KUKA KRL program: Test1.src, Test1.dat

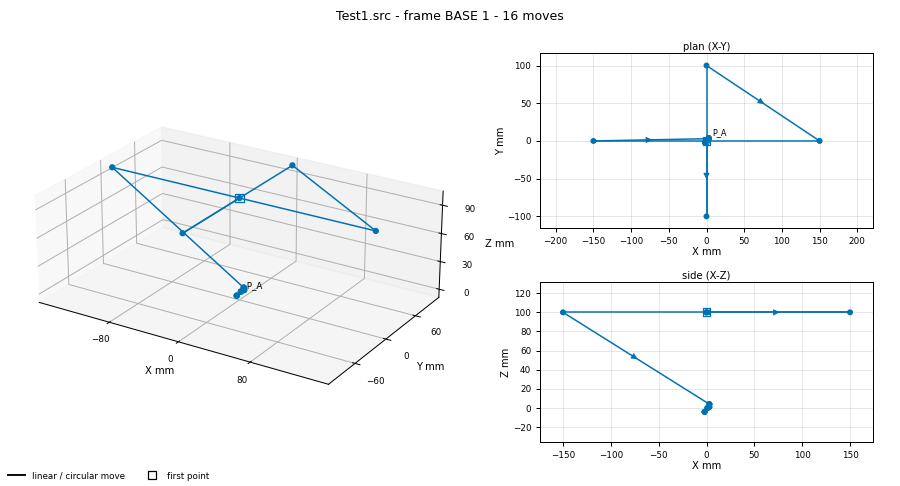
[picture p0: tool path of Test1.src in frame BASE 1, 16 of 18 moves have a stored position in this frame; points joined in program order, loops and branches not executed]
--- Test1.src ---
&ACCESS RVO1
&COMMENT Modul (src/dat) with INI line and PTP HOME at start and end of Program
DEF Test1 ( )
;FOLD INI
  ;FOLD BASISTECH INI
    GLOBAL INTERRUPT DECL 3 WHEN $STOPMESS==TRUE DO IR_STOPM ( )
    INTERRUPT ON 3
    BAS (#INITMOV,0 )
  ;ENDFOLD (BASISTECH INI)
  ;FOLD USER INI
    ;Make your modifications here

  ;ENDFOLD (USER INI)
;ENDFOLD (INI)
$TOOL = TOOL_DATA[1]
$BASE = BASE_DATA[1]

;FOLD PTP HOME  Vel= 100 % DEFAULT;%{PE}%MKUKATPBASIS,%CMOVE,%VPTP,%P 1:PTP, 2:HOME, 3:, 5:100, 7:DEFAULT
$BWDSTART = FALSE
PDAT_ACT=PDEFAULT
FDAT_ACT=FHOME
BAS (#PTP_PARAMS,100 )
$H_POS=XHOME
PTP  XHOME
;ENDFOLD

  LIN {X 0, Y 0, Z 100}
  LIN {X 0, Y -100, Z 100}
  LIN {X 0, Y 100, Z 100}
  LIN {X 150, Y 0, Z 100}
  LIN {X -150, Y 0, Z 100}

 IF mode == 1 THEN   ;IF NOT mode == 1 THEN can do it this way as well
   LIN P_A
 ELSEIF mode == 2  THEN
   LIN P_C
 ELSE
   LIN P_B
 ENDIF

   mode=2 ;change the mode during the program
 IF mode == 2 THEN
   LIN P_C
 ELSE
   LIN P_B
 ENDIF

  mode=1

 WHILE mode<4
   LIN P_A
   mode=mode + 1
 ENDWHILE

 FOR i=1 TO 3
 LIN P_D
 ENDFOR

LIN P_A
LIN P_B
LIN P_C
LIN P_D
PTP XHOME
END

--- Test1.dat ---
&ACCESS RVO1
&COMMENT Modul (src/dat) with INI line and PTP HOME at start and end of Program
DEFDAT Test1 PUBLIC

DECL INT mode = 1
DECL BOOL ready = FALSE

DECL E6POS P_A = {X 3, Y 3, Z 4, A 0, B 0, C 0}
DECL E6POS P_B = {X -2, Y -2, Z -4, A 0, B 0, C 0}
DECL E6POS P_C = {X 1, Y 1, Z 0, A 0, B 0, C 0}
DECL E6POS P_D = {X 3, Y 4, Z 1, A 0, B 0, C 0}

DECL FRAME TOOL_DATA[1]
TOOL_DATA[1] = {X 0, Y 0, Z 200, A 0, B 0, C 0}

;FOLD EXTERNAL DECLARATIONS;%{PE}%MKUKATPBASIS,%CEXT,%VCOMMON,%P
;FOLD BASISTECH EXT;%{PE}%MKUKATPBASIS,%CEXT,%VEXT,%P
EXT  BAS (BAS_COMMAND  :IN,REAL  :IN )
DECL INT SUCCESS
;ENDFOLD (BASISTECH EXT)
;FOLD USER EXT;%{E}%MKUKATPUSER,%CEXT,%VEXT,%P
;Make here your modifications

;ENDFOLD (USER EXT)
;ENDFOLD (EXTERNAL DECLERATIONS)
ENDDAT
